LIN {X 0,Y 71.337,Z 768.88,A -85,B 0,C 180,E1 -28289.511,E2 -28289.511} C_VEL
LIN {X 0,Y 69.324,Z 765.278,A -85,B 0,C 180,E1 -28300.962,E2 -28300.962} C_VEL
LIN {X 0,Y 69.422,Z 761.782,A -85,B 0,C 180,E1 -28309.101,E2 -28309.101} C_VEL
LIN {X 0,Y 70.478,Z 757.39,A -85,B 0,C 180,E1 -28317.054,E2 -28317.054} C_VEL
LIN {X 0,Y 72.906,Z 750.784,A -85,B 0,C 180,E1 -28326.145,E2 -28326.145} C_VEL
LIN {X 0,Y 76.398,Z 743.132,A -85,B 0,C 180,E1 -28333.978,E2 -28333.978} C_VEL
LIN {X 0,Y 79.45,Z 736.76,A -85,B 0,C 180,E1 -28338.96,E2 -28338.96} C_VEL
LIN {X 0,Y 80.091,Z 734.246,A -85,B 0,C 180,E1 -28340.836,E2 -28340.836} C_VEL
LIN {X 0,Y 79.689,Z 730.08,A -85,B 0,C 180,E1 -28344.147,E2 -28344.147} C_VEL
LIN {X 0,Y 79.29,Z 724.776,A -85,B 0,C 180,E1 -28348.027,E2 -28348.027} C_VEL
LIN {X 0,Y 79.728,Z 722.85,A -85,B 0,C 180,E1 -28349.133,E2 -28349.133} C_VEL
LIN {X 0,Y 79.98,Z 721.934,A -85,B 0,C 180,E1 -28349.708,E2 -28349.708} C_VEL
LIN {X 0,Y 74.87,Z 732.271,A -85,B 0,C 180,E1 -28355.384,E2 -28355.384} C_VEL
LIN {X 0,Y 69.732,Z 742.158,A -85,B 0,C 180,E1 -28363.104,E2 -28363.104} C_VEL
LIN {X 0,Y 66.404,Z 748.939,A -85,B 0,C 180,E1 -28370.385,E2 -28370.385} C_VEL
LIN {X 0,Y 63.943,Z 754.671,A -85,B 0,C 180,E1 -28378.444,E2 -28378.444} C_VEL
LIN {X 0,Y 62.32,Z 759.792,A -85,B 0,C 180,E1 -28387.868,E2 -28387.868} C_VEL
LIN {X 0,Y 62.114,Z 763.686,A -85,B 0,C 180,E1 -28397.243,E2 -28397.243} C_VEL
LIN {X 0,Y 63.149,Z 766.579,A -85,B 0,C 180,E1 -28406.188,E2 -28406.188} C_VEL
LIN {X 0,Y 65.509,Z 768.703,A -85,B 0,C 180,E1 -28414.587,E2 -28414.587} C_VEL
LIN {X 0,Y 69.052,Z 770.07,A -85,B 0,C 180,E1 -28422.221,E2 -28422.221} C_VEL
LIN {X 0,Y 73.618,Z 770.772,A -85,B 0,C 180,E1 -28428.993,E2 -28428.993} C_VEL
LIN {X 0,Y 79.004,Z 770.85,A -85,B 0,C 180,E1 -28434.896,E2 -28434.896} C_VEL
LIN {X 0,Y 85.242,Z 770.227,A -85,B 0,C 180,E1 -28440,E2 -28440} C_VEL
LIN {X 0,Y 92.081,Z 768.983,A -85,B 0,C 180,E1 -28444.377,E2 -28444.377} C_VEL
LIN {X 0,Y 103.238,Z 765.801,A -85,B 0,C 180,E1 -28449.799,E2 -28449.799} C_VEL
LIN {X 0,Y 115.295,Z 760.919,A -85,B 0,C 180,E1 -28454.112,E2 -28454.112} C_VEL
LIN {X 0,Y 116.057,Z 760.554,A -85,B 0,C 180,E1 -28454.334,E2 -28454.334} C_VEL
LIN {X 0,Y 116.658,Z 760.204,A -85,B 0,C 180,E1 -28455.446,E2 -28455.446} C_VEL
LIN {X 0,Y 117.087,Z 759.92,A -85,B 0,C 180,E1 -28457.465,E2 -28457.465} C_VEL
LIN {X 0,Y 117.189,Z 759.909,A -85,B 0,C 180,E1 -28461.09,E2 -28461.09} C_VEL
LIN {X 0,Y 116.912,Z 760.433,A -85,B 0,C 180,E1 -28465.621,E2 -28465.621} C_VEL
LIN {X 0,Y 115.494,Z 761.467,A -85,B 0,C 180,E1 -28468.077,E2 -28468.077} C_VEL
LIN {X 0,Y 106.748,Z 765.452,A -85,B 0,C 180,E1 -28471.146,E2 -28471.146} C_VEL
LIN {X 0,Y 95.397,Z 769.456,A -85,B 0,C 180,E1 -28475.87,E2 -28475.87} C_VEL
LIN {X 0,Y 85.175,Z 771.953,A -85,B 0,C 180,E1 -28482.049,E2 -28482.049} C_VEL
LIN {X 0,Y 76.217,Z 773.061,A -85,B 0,C 180,E1 -28489.802,E2 -28489.802} C_VEL
LIN {X 0,Y 69.092,Z 772.817,A -85,B 0,C 180,E1 -28499.432,E2 -28499.432} C_VEL
LIN {X 0,Y 64.622,Z 771.167,A -85,B 0,C 180,E1 -28510.96,E2 -28510.96} C_VEL
LIN {X 0,Y 63.47,Z 769.803,A -85,B 0,C 180,E1 -28517.208,E2 -28517.208} C_VEL
LIN {X 0,Y 63.081,Z 766.419,A -85,B 0,C 180,E1 -28529.205,E2 -28529.205} C_VEL
LIN {X 0,Y 62.97,Z 768.91,A -85,B 0,C 180,E1 -28536.411,E2 -28536.411} C_VEL
LIN {X 0,Y 64.724,Z 772.076,A -85,B 0,C 180,E1 -28549.014,E2 -28549.014} C_VEL
LIN {X 0,Y 69.121,Z 773.803,A -85,B 0,C 180,E1 -28560.559,E2 -28560.559} C_VEL
LIN {X 0,Y 76.278,Z 774.156,A -85,B 0,C 180,E1 -28570.165,E2 -28570.165} C_VEL
LIN {X 0,Y 85.222,Z 773.146,A -85,B 0,C 180,E1 -28577.922,E2 -28577.922} C_VEL
LIN {X 0,Y 95.403,Z 770.811,A -85,B 0,C 180,E1 -28584.13,E2 -28584.13} C_VEL
LIN {X 0,Y 106.73,Z 767.014,A -85,B 0,C 180,E1 -28588.876,E2 -28588.876} C_VEL
LIN {X 0,Y 112.602,Z 764.525,A -85,B 0,C 180,E1 -28590.906,E2 -28590.906} C_VEL
LIN {X 0,Y 114.05,Z 763.44,A -85,B 0,C 180,E1 -28594.447,E2 -28594.447} C_VEL
LIN {X 0,Y 114.945,Z 762.708,A -85,B 0,C 180,E1 -28598.478,E2 -28598.478} C_VEL
LIN {X 0,Y 115.002,Z 762.636,A -85,B 0,C 180,E1 -28602.208,E2 -28602.208} C_VEL
LIN {X 0,Y 113.563,Z 763.347,A -85,B 0,C 180,E1 -28605.668,E2 -28605.668} C_VEL
LIN {X 0,Y 105.528,Z 766.471,A -85,B 0,C 180,E1 -28608.475,E2 -28608.475} C_VEL
LIN {X 0,Y 97.929,Z 768.816,A -85,B 0,C 180,E1 -28611.748,E2 -28611.748} C_VEL
LIN {X 0,Y 90.768,Z 770.452,A -85,B 0,C 180,E1 -28615.559,E2 -28615.559} C_VEL
LIN {X 0,Y 84.136,Z 771.476,A -85,B 0,C 180,E1 -28620,E2 -28620} C_VEL
LIN {X 0,Y 77.686,Z 771.834,A -85,B 0,C 180,E1 -28625.639,E2 -28625.639} C_VEL
LIN {X 0,Y 71.968,Z 771.456,A -85,B 0,C 180,E1 -28632.425,E2 -28632.425} C_VEL
LIN {X 0,Y 67.426,Z 770.313,A -85,B 0,C 180,E1 -28640.26,E2 -28640.26} C_VEL
LIN {X 0,Y 64.225,Z 768.384,A -85,B 0,C 180,E1 -28648.901,E2 -28648.901} C_VEL
LIN {X 0,Y 62.494,Z 765.631,A -85,B 0,C 180,E1 -28658.07,E2 -28658.07} C_VEL
LIN {X 0,Y 62.385,Z 760.987,A -85,B 0,C 180,E1 -28669.854,E2 -28669.854} C_VEL
LIN {X 0,Y 63.683,Z 756.191,A -85,B 0,C 180,E1 -28678.955,E2 -28678.955} C_VEL
LIN {X 0,Y 66.102,Z 750.18,A -85,B 0,C 180,E1 -28687.728,E2 -28687.728} C_VEL
LIN {X 0,Y 69.435,Z 743.283,A -85,B 0,C 180,E1 -28695.34,E2 -28695.34} C_VEL
LIN {X 0,Y 73.981,Z 734.44,A -85,B 0,C 180,E1 -28702.492,E2 -28702.492} C_VEL
LIN {X 0,Y 78.93,Z 724.628,A -85,B 0,C 180,E1 -28708.238,E2 -28708.238} C_VEL
LIN {X 0,Y 79.728,Z 722.85,A -85,B 0,C 180,E1 -28709.133,E2 -28709.133} C_VEL
LIN {X 0,Y 79.709,Z 722.855,A -85,B 0,C 180,E1 -28709.872,E2 -28709.872} C_VEL
LIN {X 0,Y 79.088,Z 724.397,A -85,B 0,C 180,E1 -28711,E2 -28711} C_VEL
LIN {X 0,Y 76.998,Z 727.904,A -85,B 0,C 180,E1 -28712.689,E2 -28712.689} C_VEL
LIN {X 0,Y 73.455,Z 731.935,A -85,B 0,C 180,E1 -28714.61,E2 -28714.61} C_VEL
LIN {X 0,Y 65.764,Z 739.297,A -85,B 0,C 180,E1 -28718.654,E2 -28718.654} C_VEL
LIN {X 0,Y 62.667,Z 742.696,A -85,B 0,C 180,E1 -28721.828,E2 -28721.828} C_VEL
LIN {X 0,Y 62.236,Z 743.403,A -85,B 0,C 180,E1 -28722.578,E2 -28722.578} C_VEL
LIN {X 0,Y 58.745,Z 750.185,A -85,B 0,C 180,E1 -28731.03,E2 -28731.03} C_VEL
LIN {X 0,Y 55.942,Z 756.755,A -85,B 0,C 180,E1 -28742.267,E2 -28742.267} C_VEL
LIN {X 0,Y 54.973,Z 762.068,A -85,B 0,C 180,E1 -28754.67,E2 -28754.67} C_VEL
LIN {X 0,Y 55.83,Z 765.581,A -85,B 0,C 180,E1 -28765.499,E2 -28765.499} C_VEL
LIN {X 0,Y 59.978,Z 769.007,A -85,B 0,C 180,E1 -28779.613,E2 -28779.613} C_VEL
LIN {X 0,Y 64.646,Z 770.427,A -85,B 0,C 180,E1 -28788.067,E2 -28788.067} C_VEL
LIN {X 0,Y 70.51,Z 771.064,A -85,B 0,C 180,E1 -28795.341,E2 -28795.341} C_VEL
LIN {X 0,Y 77.327,Z 770.958,A -85,B 0,C 180,E1 -28801.394,E2 -28801.394} C_VEL
LIN {X 0,Y 84.851,Z 770.124,A -85,B 0,C 180,E1 -28806.334,E2 -28806.334} C_VEL
LIN {X 0,Y 92.897,Z 768.516,A -85,B 0,C 180,E1 -28810.435,E2 -28810.435} C_VEL
LIN {X 0,Y 101.332,Z 766.144,A -85,B 0,C 180,E1 -28813.844,E2 -28813.844} C_VEL
LIN {X 0,Y 110.025,Z 762.999,A -85,B 0,C 180,E1 -28816.642,E2 -28816.642} C_VEL
LIN {X 0,Y 110.54,Z 762.772,A -85,B 0,C 180,E1 -28817.514,E2 -28817.514} C_VEL
LIN {X 0,Y 110.567,Z 762.896,A -85,B 0,C 180,E1 -28822.419,E2 -28822.419} C_VEL
LIN {X 0,Y 109.348,Z 763.697,A -85,B 0,C 180,E1 -28825.871,E2 -28825.871} C_VEL
LIN {X 0,Y 100.245,Z 767.168,A -85,B 0,C 180,E1 -28828.799,E2 -28828.799} C_VEL
LIN {X 0,Y 91.428,Z 769.791,A -85,B 0,C 180,E1 -28832.272,E2 -28832.272} C_VEL
LIN {X 0,Y 80.584,Z 772.023,A -85,B 0,C 180,E1 -28838.291,E2 -28838.291} C_VEL
LIN {X 0,Y 70.924,Z 772.909,A -85,B 0,C 180,E1 -28846.084,E2 -28846.084} C_VEL
LIN {X 0,Y 63.07,Z 772.384,A -85,B 0,C 180,E1 -28856.144,E2 -28856.144} C_VEL
LIN {X 0,Y 57.958,Z 770.51,A -85,B 0,C 180,E1 -28868.671,E2 -28868.671} C_VEL
LIN {X 0,Y 56.601,Z 769.057,A -85,B 0,C 180,E1 -28875.624,E2 -28875.624} C_VEL
LIN {X 0,Y 56.083,Z 765.346,A -85,B 0,C 180,E1 -28889.106,E2 -28889.106} C_VEL
LIN {X 0,Y 55.97,Z 768.007,A -85,B 0,C 180,E1 -28897.217,E2 -28897.217} C_VEL
LIN {X 0,Y 56.623,Z 769.911,A -85,B 0,C 180,E1 -28904.376,E2 -28904.376} C_VEL
LIN {X 0,Y 60.188,Z 772.525,A -85,B 0,C 180,E1 -28917.847,E2 -28917.847} C_VEL
LIN {X 0,Y 66.808,Z 773.802,A -85,B 0,C 180,E1 -28929.14,E2 -28929.14} C_VEL
LIN {X 0,Y 75.603,Z 773.75,A -85,B 0,C 180,E1 -28938.048,E2 -28938.048} C_VEL
LIN {X 0,Y 85.892,Z 772.333,A -85,B 0,C 180,E1 -28944.912,E2 -28944.912} C_VEL
LIN {X 0,Y 97.253,Z 769.539,A -85,B 0,C 180,E1 -28950.136,E2 -28950.136} C_VEL
LIN {X 0,Y 106.304,Z 766.519,A -85,B 0,C 180,E1 -28953.193,E2 -28953.193} C_VEL
LIN {X 0,Y 107.731,Z 765.731,A -85,B 0,C 180,E1 -28955.971,E2 -28955.971} C_VEL
LIN {X 0,Y 108.018,Z 765.544,A -85,B 0,C 180,E1 -28957.022,E2 -28957.022} C_VEL
LIN {X 0,Y 108.329,Z 765.267,A -85,B 0,C 180,E1 -28961.072,E2 -28961.072} C_VEL
LIN {X 0,Y 107.845,Z 765.438,A -85,B 0,C 180,E1 -28962.947,E2 -28962.947} C_VEL
LIN {X 0,Y 101.776,Z 767.468,A -85,B 0,C 180,E1 -28965.189,E2 -28965.189} C_VEL
LIN {X 0,Y 93.203,Z 769.734,A -85,B 0,C 180,E1 -28968.607,E2 -28968.607} C_VEL
LIN {X 0,Y 81.279,Z 771.719,A -85,B 0,C 180,E1 -28975.04,E2 -28975.04} C_VEL
LIN {X 0,Y 74.635,Z 772.074,A -85,B 0,C 180,E1 -28980,E2 -28980} C_VEL
LIN {X 0,Y 68.707,Z 771.862,A -85,B 0,C 180,E1 -28985.871,E2 -28985.871} C_VEL
LIN {X 0,Y 63.649,Z 770.982,A -85,B 0,C 180,E1 -28992.758,E2 -28992.758} C_VEL
LIN {X 0,Y 57.995,Z 768.511,A -85,B 0,C 180,E1 -29005.097,E2 -29005.097} C_VEL
LIN {X 0,Y 55.23,Z 764.137,A -85,B 0,C 180,E1 -29020.223,E2 -29020.223} C_VEL
LIN {X 0,Y 55.62,Z 759.061,A -85,B 0,C 180,E1 -29033.115,E2 -29033.115} C_VEL
LIN {X 0,Y 57.844,Z 752.738,A -85,B 0,C 180,E1 -29044.83,E2 -29044.83} C_VEL
LIN {X 0,Y 61.613,Z 745.011,A -85,B 0,C 180,E1 -29055.126,E2 -29055.126} C_VEL
LIN {X 0,Y 66.169,Z 736.739,A -85,B 0,C 180,E1 -29063.005,E2 -29063.005} C_VEL
LIN {X 0,Y 71.341,Z 727.085,A -85,B 0,C 180,E1 -29069.575,E2 -29069.575} C_VEL
LIN {X 0,Y 65.022,Z 738.266,A -85,B 0,C 180,E1 -29077.615,E2 -29077.615} C_VEL
LIN {X 0,Y 62.236,Z 743.403,A -85,B 0,C 180,E1 -29082.578,E2 -29082.578} C_VEL
LIN {X 0,Y 59.725,Z 746.862,A -85,B 0,C 180,E1 -29086.416,E2 -29086.416} C_VEL
LIN {X 0,Y 54.307,Z 751.878,A -85,B 0,C 180,E1 -29093.106,E2 -29093.106} C_VEL
LIN {X 0,Y 49.514,Z 756.287,A -85,B 0,C 180,E1 -29101.51,E2 -29101.51} C_VEL
LIN {X 0,Y 48.175,Z 758.808,A -85,B 0,C 180,E1 -29107.661,E2 -29107.661} C_VEL
LIN {X 0,Y 48.163,Z 763.325,A -85,B 0,C 180,E1 -29120.915,E2 -29120.915} C_VEL
LIN {X 0,Y 50.899,Z 767.174,A -85,B 0,C 180,E1 -29135.529,E2 -29135.529} C_VEL
LIN {X 0,Y 57.195,Z 769.99,A -85,B 0,C 180,E1 -29149.408,E2 -29149.408} C_VEL
LIN {X 0,Y 65.904,Z 771.234,A -85,B 0,C 180,E1 -29160,E2 -29160} C_VEL
LIN {X 0,Y 72.751,Z 771.307,A -85,B 0,C 180,E1 -29165.543,E2 -29165.543} C_VEL
LIN {X 0,Y 80.268,Z 770.682,A -85,B 0,C 180,E1 -29170.085,E2 -29170.085} C_VEL
LIN {X 0,Y 88.229,Z 769.438,A -85,B 0,C 180,E1 -29173.826,E2 -29173.826} C_VEL
LIN {X 0,Y 100.893,Z 766.228,A -85,B 0,C 180,E1 -29178.268,E2 -29178.268} C_VEL
LIN {X 0,Y 103.865,Z 765.283,A -85,B 0,C 180,E1 -29179.775,E2 -29179.775} C_VEL
LIN {X 0,Y 103.031,Z 765.767,A -85,B 0,C 180,E1 -29183.41,E2 -29183.41} C_VEL
LIN {X 0,Y 93.933,Z 768.591,A -85,B 0,C 180,E1 -29186.131,E2 -29186.131} C_VEL
LIN {X 0,Y 81.977,Z 771.274,A -85,B 0,C 180,E1 -29190.989,E2 -29190.989} C_VEL
LIN {X 0,Y 71.017,Z 772.534,A -85,B 0,C 180,E1 -29197.66,E2 -29197.66} C_VEL
LIN {X 0,Y 61.386,Z 772.456,A -85,B 0,C 180,E1 -29206.617,E2 -29206.617} C_VEL
LIN {X 0,Y 53.982,Z 771.053,A -85,B 0,C 180,E1 -29218.62,E2 -29218.62} C_VEL
LIN {X 0,Y 49.792,Z 768.227,A -85,B 0,C 180,E1 -29233.606,E2 -29233.606} C_VEL
LIN {X 0,Y 49.059,Z 764.257,A -85,B 0,C 180,E1 -29248.977,E2 -29248.977} C_VEL
LIN {X 0,Y 49.273,Z 768.08,A -85,B 0,C 180,E1 -29262.358,E2 -29262.358} C_VEL
LIN {X 0,Y 51.547,Z 770.652,A -85,B 0,C 180,E1 -29274.147,E2 -29274.147} C_VEL
LIN {X 0,Y 57.339,Z 772.841,A -85,B 0,C 180,E1 -29287.799,E2 -29287.799} C_VEL
LIN {X 0,Y 66.032,Z 773.671,A -85,B 0,C 180,E1 -29298.166,E2 -29298.166} C_VEL
LIN {X 0,Y 76.424,Z 773.189,A -85,B 0,C 180,E1 -29305.862,E2 -29305.862} C_VEL
LIN {X 0,Y 87.853,Z 771.401,A -85,B 0,C 180,E1 -29311.642,E2 -29311.642} C_VEL
LIN {X 0,Y 100.151,Z 768.209,A -85,B 0,C 180,E1 -29315.823,E2 -29315.823} C_VEL
LIN {X 0,Y 101.424,Z 767.598,A -85,B 0,C 180,E1 -29319.729,E2 -29319.729} C_VEL
LIN {X 0,Y 95.025,Z 769.295,A -85,B 0,C 180,E1 -29322.792,E2 -29322.792} C_VEL
LIN {X 0,Y 86.845,Z 770.938,A -85,B 0,C 180,E1 -29325.95,E2 -29325.95} C_VEL
LIN {X 0,Y 78.482,Z 772.013,A -85,B 0,C 180,E1 -29330.088,E2 -29330.088} C_VEL
LIN {X 0,Y 70.519,Z 772.335,A -85,B 0,C 180,E1 -29335.307,E2 -29335.307} C_VEL
LIN {X 0,Y 63.289,Z 771.897,A -85,B 0,C 180,E1 -29341.876,E2 -29341.876} C_VEL
LIN {X 0,Y 57.103,Z 770.711,A -85,B 0,C 180,E1 -29350.051,E2 -29350.051} C_VEL
LIN {X 0,Y 52.295,Z 768.758,A -85,B 0,C 180,E1 -29359.816,E2 -29359.816} C_VEL
LIN {X 0,Y 48.53,Z 764.728,A -85,B 0,C 180,E1 -29375.4,E2 -29375.4} C_VEL
LIN {X 0,Y 48.312,Z 759.538,A -85,B 0,C 180,E1 -29390.899,E2 -29390.899} C_VEL
LIN {X 0,Y 49.928,Z 754.516,A -85,B 0,C 180,E1 -29402.167,E2 -29402.167} C_VEL
LIN {X 0,Y 52.932,Z 748.24,A -85,B 0,C 180,E1 -29412.732,E2 -29412.732} C_VEL
LIN {X 0,Y 56.893,Z 741.334,A -85,B 0,C 180,E1 -29421.211,E2 -29421.211} C_VEL
LIN {X 0,Y 62.327,Z 732.188,A -85,B 0,C 180,E1 -29429.19,E2 -29429.19} C_VEL
LIN {X 0,Y 62.459,Z 731.607,A -85,B 0,C 180,E1 -29429.695,E2 -29429.695} C_VEL
LIN {X 0,Y 56.769,Z 741.056,A -85,B 0,C 180,E1 -29437.943,E2 -29437.943} C_VEL
LIN {X 0,Y 52.618,Z 748.32,A -85,B 0,C 180,E1 -29447.078,E2 -29447.078} C_VEL
LIN {X 0,Y 49.654,Z 754.427,A -85,B 0,C 180,E1 -29457.657,E2 -29457.657} C_VEL
LIN {X 0,Y 48.175,Z 758.808,A -85,B 0,C 180,E1 -29467.661,E2 -29467.661} C_VEL
LIN {X 0,Y 47.291,Z 761.108,A -85,B 0,C 180,E1 -29474.095,E2 -29474.095} C_VEL
LIN {X 0,Y 45.168,Z 764.209,A -85,B 0,C 180,E1 -29485.486,E2 -29485.486} C_VEL
LIN {X 0,Y 44.6,Z 766.216,A -85,B 0,C 180,E1 -29495.372,E2 -29495.372} C_VEL
LIN {X 0,Y 45.791,Z 767.582,A -85,B 0,C 180,E1 -29502.587,E2 -29502.587} C_VEL
LIN {X 0,Y 46.589,Z 767.975,A -85,B 0,C 180,E1 -29504.783,E2 -29504.783} C_VEL
LIN {X 0,Y 50.283,Z 769.453,A -85,B 0,C 180,E1 -29511.965,E2 -29511.965} C_VEL
LIN {X 0,Y 56.309,Z 770.785,A -85,B 0,C 180,E1 -29520,E2 -29520} C_VEL
LIN {X 0,Y 63.702,Z 771.488,A -85,B 0,C 180,E1 -29526.839,E2 -29526.839} C_VEL
LIN {X 0,Y 71.882,Z 771.482,A -85,B 0,C 180,E1 -29532.132,E2 -29532.132} C_VEL
LIN {X 0,Y 80.513,Z 770.74,A -85,B 0,C 180,E1 -29536.23,E2 -29536.23} C_VEL
LIN {X 0,Y 93.557,Z 768.356,A -85,B 0,C 180,E1 -29540.773,E2 -29540.773} C_VEL
LIN {X 0,Y 91.035,Z 769.034,A -85,B 0,C 180,E1 -29542.123,E2 -29542.123} C_VEL
LIN {X 0,Y 78.205,Z 771.424,A -85,B 0,C 180,E1 -29546.701,E2 -29546.701} C_VEL
LIN {X 0,Y 66.915,Z 772.393,A -85,B 0,C 180,E1 -29552.841,E2 -29552.841} C_VEL
LIN {X 0,Y 56.43,Z 772.081,A -85,B 0,C 180,E1 -29561.651,E2 -29561.651} C_VEL
LIN {X 0,Y 48.067,Z 770.39,A -85,B 0,C 180,E1 -29574.213,E2 -29574.213} C_VEL
LIN {X 0,Y 43.066,Z 767.342,A -85,B 0,C 180,E1 -29590.955,E2 -29590.955} C_VEL
LIN {X 0,Y 42.062,Z 763.107,A -85,B 0,C 180,E1 -29609.107,E2 -29609.107} C_VEL
LIN {X 0,Y 42.451,Z 767.071,A -85,B 0,C 180,E1 -29624.383,E2 -29624.383} C_VEL
LIN {X 0,Y 45.185,Z 769.845,A -85,B 0,C 180,E1 -29637.819,E2 -29637.819} C_VEL
LIN {X 0,Y 51.915,Z 772.252,A -85,B 0,C 180,E1 -29652.604,E2 -29652.604} C_VEL
LIN {X 0,Y 61.512,Z 773.376,A -85,B 0,C 180,E1 -29663.113,E2 -29663.113} C_VEL
LIN {X 0,Y 72.664,Z 773.155,A -85,B 0,C 180,E1 -29670.518,E2 -29670.518} C_VEL
LIN {X 0,Y 84.71,Z 771.614,A -85,B 0,C 180,E1 -29675.874,E2 -29675.874} C_VEL
LIN {X 0,Y 91.037,Z 770.341,A -85,B 0,C 180,E1 -29677.884,E2 -29677.884} C_VEL
LIN {X 0,Y 91.711,Z 770.148,A -85,B 0,C 180,E1 -29678.976,E2 -29678.976} C_VEL
LIN {X 0,Y 80.944,Z 771.87,A -85,B 0,C 180,E1 -29682.767,E2 -29682.767} C_VEL
LIN {X 0,Y 69.678,Z 772.571,A -85,B 0,C 180,E1 -29688.362,E2 -29688.362} C_VEL
LIN {X 0,Y 62.293,Z 772.356,A -85,B 0,C 180,E1 -29693.522,E2 -29693.522} C_VEL
LIN {X 0,Y 55.626,Z 771.484,A -85,B 0,C 180,E1 -29700,E2 -29700} C_VEL
LIN {X 0,Y 47.331,Z 769.062,A -85,B 0,C 180,E1 -29712.865,E2 -29712.865} C_VEL
LIN {X 0,Y 42.117,Z 765.069,A -85,B 0,C 180,E1 -29730.04,E2 -29730.04} C_VEL
LIN {X 0,Y 41.042,Z 760.339,A -85,B 0,C 180,E1 -29746.762,E2 -29746.762} C_VEL
LIN {X 0,Y 42.86,Z 754.21,A -85,B 0,C 180,E1 -29763.085,E2 -29763.085} C_VEL
LIN {X 0,Y 46.853,Z 746.667,A -85,B 0,C 180,E1 -29776.993,E2 -29776.993} C_VEL
LIN {X 0,Y 52.098,Z 738.445,A -85,B 0,C 180,E1 -29787.097,E2 -29787.097} C_VEL
LIN {X 0,Y 53.573,Z 735.891,A -85,B 0,C 180,E1 -29789.644,E2 -29789.644} C_VEL
LIN {X 0,Y 47.44,Z 745.332,A -85,B 0,C 180,E1 -29800.668,E2 -29800.668} C_VEL
LIN {X 0,Y 43.137,Z 752.896,A -85,B 0,C 180,E1 -29814.026,E2 -29814.026} C_VEL
LIN {X 0,Y 41.104,Z 758.218,A -85,B 0,C 180,E1 -29827.429,E2 -29827.429} C_VEL
LIN {X 0,Y 41.207,Z 762.766,A -85,B 0,C 180,E1 -29842.434,E2 -29842.434} C_VEL
LIN {X 0,Y 44.814,Z 767.053,A -85,B 0,C 180,E1 -29860.201,E2 -29860.201} C_VEL
LIN {X 0,Y 46.589,Z 767.975,A -85,B 0,C 180,E1 -29864.783,E2 -29864.783} C_VEL
LIN {X 0,Y 48.975,Z 769.19,A -85,B 0,C 180,E1 -29871.131,E2 -29871.131} C_VEL
LIN {X 0,Y 52.656,Z 770.583,A -85,B 0,C 180,E1 -29881.425,E2 -29881.425} C_VEL
LIN {X 0,Y 57.846,Z 771.468,A -85,B 0,C 180,E1 -29890.173,E2 -29890.173} C_VEL
LIN {X 0,Y 62.271,Z 771.718,A -85,B 0,C 180,E1 -29893.91,E2 -29893.91} C_VEL
LIN {X 0,Y 74.711,Z 771.494,A -85,B 0,C 180,E1 -29899.839,E2 -29899.839} C_VEL
LIN {X 0,Y 76.324,Z 771.354,A -85,B 0,C 180,E1 -29900.459,E2 -29900.459} C_VEL
LIN {X 0,Y 75.649,Z 771.48,A -85,B 0,C 180,E1 -29901.724,E2 -29901.724} C_VEL
LIN {X 0,Y 63.346,Z 772.205,A -85,B 0,C 180,E1 -29907.438,E2 -29907.438} C_VEL
LIN {X 0,Y 51.978,Z 771.6,A -85,B 0,C 180,E1 -29915.786,E2 -29915.786} C_VEL
LIN {X 0,Y 42.518,Z 769.694,A -85,B 0,C 180,E1 -29928.616,E2 -29928.616} C_VEL
LIN {X 0,Y 36.469,Z 766.397,A -85,B 0,C 180,E1 -29947.335,E2 -29947.335} C_VEL
LIN {X 0,Y 35.095,Z 761.855,A -85,B 0,C 180,E1 -29968.929,E2 -29968.929} C_VEL
LIN {X 0,Y 35.692,Z 766.026,A -85,B 0,C 180,E1 -29987.184,E2 -29987.184} C_VEL
LIN {X 0,Y 39.071,Z 768.979,A -85,B 0,C 180,E1 -30002.664,E2 -30002.664} C_VEL
LIN {X 0,Y 46.942,Z 771.641,A -85,B 0,C 180,E1 -30018.473,E2 -30018.473} C_VEL
LIN {X 0,Y 57.525,Z 772.985,A -85,B 0,C 180,E1 -30028.788,E2 -30028.788} C_VEL
LIN {X 0,Y 69.436,Z 773.042,A -85,B 0,C 180,E1 -30035.641,E2 -30035.641} C_VEL
LIN {X 0,Y 75.667,Z 772.586,A -85,B 0,C 180,E1 -30038.255,E2 -30038.255} C_VEL
LIN {X 0,Y 75.211,Z 772.581,A -85,B 0,C 180,E1 -30039.143,E2 -30039.143} C_VEL
LIN {X 0,Y 66.079,Z 772.839,A -85,B 0,C 180,E1 -30043.187,E2 -30043.187} C_VEL
LIN {X 0,Y 57.351,Z 772.312,A -85,B 0,C 180,E1 -30048.636,E2 -30048.636} C_VEL
LIN {X 0,Y 46.119,Z 770.28,A -85,B 0,C 180,E1 -30060,E2 -30060} C_VEL
LIN {X 0,Y 40.383,Z 768.155,A -85,B 0,C 180,E1 -30070.023,E2 -30070.023} C_VEL
LIN {X 0,Y 35.054,Z 764.021,A -85,B 0,C 180,E1 -30088.805,E2 -30088.805} C_VEL
LIN {X 0,Y 33.957,Z 760.018,A -85,B 0,C 180,E1 -30105,E2 -30105} C_VEL
LIN {X 0,Y 35.772,Z 753.922,A -85,B 0,C 180,E1 -30124.298,E2 -30124.298} C_VEL
LIN {X 0,Y 40.043,Z 746.558,A -85,B 0,C 180,E1 -30139.887,E2 -30139.887} C_VEL
LIN {X 0,Y 44.771,Z 739.789,A -85,B 0,C 180,E1 -30149.408,E2 -30149.408} C_VEL
LIN {X 0,Y 44.462,Z 739.806,A -85,B 0,C 180,E1 -30149.996,E2 -30149.996} C_VEL
LIN {X 0,Y 39.635,Z 746.804,A -85,B 0,C 180,E1 -30160.209,E2 -30160.209} C_VEL
LIN {X 0,Y 35.414,Z 753.873,A -85,B 0,C 180,E1 -30175.812,E2 -30175.812} C_VEL
LIN {X 0,Y 33.8,Z 759.737,A -85,B 0,C 180,E1 -30194.998,E2 -30194.998} C_VEL
LIN {X 0,Y 36.313,Z 764.964,A -85,B 0,C 180,E1 -30217.227,E2 -30217.227} C_VEL
LIN {X 0,Y 42.44,Z 768.392,A -85,B 0,C 180,E1 -30233.474,E2 -30233.474} C_VEL
LIN {X 0,Y 49.27,Z 770.27,A -85,B 0,C 180,E1 -30243.206,E2 -30243.206} C_VEL
LIN {X 0,Y 61.226,Z 771.689,A -85,B 0,C 180,E1 -30253.272,E2 -30253.272} C_VEL
LIN {X 0,Y 62.271,Z 771.718,A -85,B 0,C 180,E1 -30253.91,E2 -30253.91} C_VEL
LIN {X 0,Y 62.87,Z 771.786,A -85,B 0,C 180,E1 -30255.096,E2 -30255.096} C_VEL
LIN {X 0,Y 62.2,Z 771.855,A -85,B 0,C 180,E1 -30257.454,E2 -30257.454} C_VEL
LIN {X 0,Y 59.293,Z 771.905,A -85,B 0,C 180,E1 -30260.851,E2 -30260.851} C_VEL
LIN {X 0,Y 56.525,Z 771.812,A -85,B 0,C 180,E1 -30263.087,E2 -30263.087} C_VEL
LIN {X 0,Y 47.442,Z 771.011,A -85,B 0,C 180,E1 -30269.698,E2 -30269.698} C_VEL
LIN {X 0,Y 39.105,Z 769.339,A -85,B 0,C 180,E1 -30278.85,E2 -30278.85} C_VEL
LIN {X 0,Y 33.226,Z 767.309,A -85,B 0,C 180,E1 -30290.62,E2 -30290.62} C_VEL
LIN {X 0,Y 28.315,Z 763.018,A -85,B 0,C 180,E1 -30315.635,E2 -30315.635} C_VEL
LIN {X 0,Y 28.117,Z 760.526,A -85,B 0,C 180,E1 -30328.887,E2 -30328.887} C_VEL
LIN {X 0,Y 29.072,Z 764.865,A -85,B 0,C 180,E1 -30351.267,E2 -30351.267} C_VEL
LIN {X 0,Y 33.34,Z 768.019,A -85,B 0,C 180,E1 -30369.233,E2 -30369.233} C_VEL
LIN {X 0,Y 42.578,Z 770.94,A -85,B 0,C 180,E1 -30385.626,E2 -30385.626} C_VEL
LIN {X 0,Y 54.183,Z 772.579,A -85,B 0,C 180,E1 -30395.232,E2 -30395.232} C_VEL
LIN {X 0,Y 60.429,Z 772.903,A -85,B 0,C 180,E1 -30398.505,E2 -30398.505} C_VEL
LIN {X 0,Y 51.167,Z 771.946,A -85,B 0,C 180,E1 -30404.056,E2 -30404.056} C_VEL
LIN {X 0,Y 42.623,Z 770.264,A -85,B 0,C 180,E1 -30411.642,E2 -30411.642} C_VEL
LIN {X 0,Y 33.136,Z 766.851,A -85,B 0,C 180,E1 -30427.143,E2 -30427.143} C_VEL
LIN {X 0,Y 27.605,Z 762.098,A -85,B 0,C 180,E1 -30450.61,E2 -30450.61} C_VEL
LIN {X 0,Y 27.367,Z 756.542,A -85,B 0,C 180,E1 -30475.408,E2 -30475.408} C_VEL
LIN {X 0,Y 30.372,Z 750.746,A -85,B 0,C 180,E1 -30494.136,E2 -30494.136} C_VEL
LIN {X 0,Y 35.803,Z 743.263,A -85,B 0,C 180,E1 -30509.417,E2 -30509.417} C_VEL
LIN {X 0,Y 35.595,Z 743.185,A -85,B 0,C 180,E1 -30509.995,E2 -30509.995} C_VEL
LIN {X 0,Y 30.674,Z 749.725,A -85,B 0,C 180,E1 -30523.239,E2 -30523.239} C_VEL
LIN {X 0,Y 27.452,Z 755.341,A -85,B 0,C 180,E1 -30540.791,E2 -30540.791} C_VEL
LIN {X 0,Y 26.927,Z 760.119,A -85,B 0,C 180,E1 -30561.525,E2 -30561.525} C_VEL
LIN {X 0,Y 31.249,Z 765.217,A -85,B 0,C 180,E1 -30587.002,E2 -30587.002} C_VEL
LIN {X 0,Y 36.98,Z 767.871,A -85,B 0,C 180,E1 -30600,E2 -30600} C_VEL
LIN {X 0,Y 44.067,Z 769.879,A -85,B 0,C 180,E1 -30609.177,E2 -30609.177} C_VEL
LIN {X 0,Y 51.911,Z 771.208,A -85,B 0,C 180,E1 -30615.71,E2 -30615.71} C_VEL
LIN {X 0,Y 60.284,Z 771.914,A -85,B 0,C 180,E1 -30620.471,E2 -30620.471} C_VEL
LIN {X 0,Y 60.405,Z 771.948,A -85,B 0,C 180,E1 -30621.451,E2 -30621.451} C_VEL
LIN {X 0,Y 48.169,Z 771.111,A -85,B 0,C 180,E1 -30628.914,E2 -30628.914} C_VEL
LIN {X 0,Y 39.105,Z 769.339,A -85,B 0,C 180,E1 -30638.85,E2 -30638.85} C_VEL
LIN {X 0,Y 34.883,Z 768.12,A -85,B 0,C 180,E1 -30644.943,E2 -30644.943} C_VEL
LIN {X 0,Y 27.785,Z 765.247,A -85,B 0,C 180,E1 -30656.491,E2 -30656.491} C_VEL
LIN {X 0,Y 23.137,Z 762.402,A -85,B 0,C 180,E1 -30669.71,E2 -30669.71} C_VEL
LIN {X 0,Y 21.175,Z 759.166,A -85,B 0,C 180,E1 -30687.923,E2 -30687.923} C_VEL
LIN {X 0,Y 22.692,Z 763.667,A -85,B 0,C 180,E1 -30717.69,E2 -30717.69} C_VEL
LIN {X 0,Y 28.224,Z 767.012,A -85,B 0,C 180,E1 -30738.341,E2 -30738.341} C_VEL
LIN {X 0,Y 39.023,Z 770.183,A -85,B 0,C 180,E1 -30754.231,E2 -30754.231} C_VEL
LIN {X 0,Y 41.007,Z 770.576,A -85,B 0,C 180,E1 -30755.835,E2 -30755.835} C_VEL
LIN {X 0,Y 43.742,Z 771.041,A -85,B 0,C 180,E1 -30759.357,E2 -30759.357} C_VEL
LIN {X 0,Y 31.015,Z 767.502,A -85,B 0,C 180,E1 -30772.454,E2 -30772.454} C_VEL
LIN {X 0,Y 22.09,Z 762.593,A -85,B 0,C 180,E1 -30797.331,E2 -30797.331} C_VEL
LIN {X 0,Y 20.074,Z 756.678,A -85,B 0,C 180,E1 -30832.206,E2 -30832.206} C_VEL
LIN {X 0,Y 23.194,Z 750.926,A -85,B 0,C 180,E1 -30857.041,E2 -30857.041} C_VEL
LIN {X 0,Y 25.583,Z 747.851,A -85,B 0,C 180,E1 -30866.055,E2 -30866.055} C_VEL
LIN {X 0,Y 26.508,Z 746.375,A -85,B 0,C 180,E1 -30870.231,E2 -30870.231} C_VEL
LIN {X 0,Y 21.702,Z 752.44,A -85,B 0,C 180,E1 -30888.887,E2 -30888.887} C_VEL
LIN {X 0,Y 19.74,Z 757.721,A -85,B 0,C 180,E1 -30915.388,E2 -30915.388} C_VEL
LIN {X 0,Y 22.092,Z 762.162,A -85,B 0,C 180,E1 -30942.6,E2 -30942.6} C_VEL
LIN {X 0,Y 28.121,Z 765.757,A -85,B 0,C 180,E1 -30961.655,E2 -30961.655} C_VEL
LIN {X 0,Y 36.129,Z 768.522,A -85,B 0,C 180,E1 -30973.458,E2 -30973.458} C_VEL
LIN {X 0,Y 45.169,Z 770.506,A -85,B 0,C 180,E1 -30981.015,E2 -30981.015} C_VEL
LIN {X 0,Y 33.235,Z 768.076,A -85,B 0,C 180,E1 -30992.245,E2 -30992.245} C_VEL
LIN {X 0,Y 24.087,Z 764.267,A -85,B 0,C 180,E1 -31014.308,E2 -31014.308} C_VEL
LIN {X 0,Y 21.175,Z 759.166,A -85,B 0,C 180,E1 -31047.923,E2 -31047.923} C_VEL
LIN {X 0,Y 20.617,Z 760.519,A -85,B 0,C 180,E1 -31057.961,E2 -31057.961} C_VEL
LIN {X 0,Y 19.616,Z 761.634,A -85,B 0,C 180,E1 -31068.513,E2 -31068.513} C_VEL
LIN {X 0,Y 19.371,Z 763.932,A -85,B 0,C 180,E1 -31095.993,E2 -31095.993} C_VEL
LIN {X 0,Y 21.497,Z 764.856,A -85,B 0,C 180,E1 -31105.418,E2 -31105.418} C_VEL
LIN {X 0,Y 24.132,Z 765.884,A -85,B 0,C 180,E1 -31110.906,E2 -31110.906} C_VEL
LIN {X 0,Y 27.679,Z 767.03,A -85,B 0,C 180,E1 -31120.189,E2 -31120.189} C_VEL
LIN {X 0,Y 17.591,Z 762.568,A -85,B 0,C 180,E1 -31140.001,E2 -31140.001} C_VEL
LIN {X 0,Y 12.899,Z 756.773,A -85,B 0,C 180,E1 -31185.033,E2 -31185.033} C_VEL
LIN {X 0,Y 16.122,Z 751.043,A -85,B 0,C 180,E1 -31222.633,E2 -31222.633} C_VEL
LIN {X 0,Y 17.391,Z 749.327,A -85,B 0,C 180,E1 -31229.99,E2 -31229.99} C_VEL
LIN {X 0,Y 12.736,Z 756.455,A -85,B 0,C 180,E1 -31274.94,E2 -31274.94} C_VEL
LIN {X 0,Y 17.688,Z 762.157,A -85,B 0,C 180,E1 -31319.999,E2 -31319.999} C_VEL
LIN {X 0,Y 27.945,Z 766.495,A -85,B 0,C 180,E1 -31339.465,E2 -31339.465} C_VEL
LIN {X 0,Y 24.06,Z 765.288,A -85,B 0,C 180,E1 -31348.815,E2 -31348.815} C_VEL
LIN {X 0,Y 15.188,Z 760.445,A -85,B 0,C 180,E1 -31382.448,E2 -31382.448} C_VEL
LIN {X 0,Y 14.216,Z 757.699,A -85,B 0,C 180,E1 -31409.039,E2 -31409.039} C_VEL
LIN {X 0,Y 16.842,Z 762.335,A -85,B 0,C 180,E1 -31448.764,E2 -31448.764} C_VEL
LIN {X 0,Y 21.497,Z 764.856,A -85,B 0,C 180,E1 -31465.418,E2 -31465.418} C_VEL
LIN {X 0,Y 20.09,Z 764.517,A -85,B 0,C 180,E1 -31465.898,E2 -31465.898} C_VEL
LIN {X 0,Y 14.129,Z 762.649,A -85,B 0,C 180,E1 -31456.29,E2 -31456.29} C_VEL
LIN {X 0,Y 8.246,Z 759.927,A -85,B 0,C 180,E1 -31397.154,E2 -31397.154} C_VEL
LIN {X 0,Y 9.825,Z 759.744,A -85,B 0,C 180,E1 -31363.901,E2 -31363.901} C_VEL
LIN {X 0,Y 12.121,Z 760.45,A -85,B 0,C 180,E1 -31346.941,E2 -31346.941} C_VEL
LIN {X 0,Y 13.392,Z 761.013,A -85,B 0,C 180,E1 -31340.789,E2 -31340.789} C_VEL
LIN {X 0,Y 5.765,Z 754.924,A -85,B 0,C 180,E1 -31270.562,E2 -31270.562} C_VEL
LIN {X 0,Y 7.869,Z 752.167,A -85,B 0,C 180,E1 -31229.978,E2 -31229.978} C_VEL
LIN {X 0,Y 7.158,Z 753.17,A -85,B 0,C 180,E1 -31219.074,E2 -31219.074} C_VEL
LIN {X 0,Y 9.757,Z 759.568,A -85,B 0,C 180,E1 -31130.276,E2 -31130.276} C_VEL
LIN {X 0,Y 13.396,Z 761.483,A -85,B 0,C 180,E1 -31118.921,E2 -31118.921} C_VEL
LIN {X 0,Y 11.068,Z 760.351,A -85,B 0,C 180,E1 -31105.056,E2 -31105.056} C_VEL
LIN {X 0,Y 7.338,Z 756.014,A -85,B 0,C 180,E1 -31046.252,E2 -31046.252} C_VEL
LIN {X 0,Y 11.005,Z 759.878,A -85,B 0,C 180,E1 -30994.556,E2 -30994.556} C_VEL
LIN {X 0,Y 12.121,Z 760.45,A -85,B 0,C 180,E1 -30986.941,E2 -30986.941} C_VEL
LIN {X 0,Y 12.121,Z 760.45,A -85,B 0,C 180,E1 -30986.941,E2 -30986.941}

QRS_NEXT_CUT()

QRS_NEXT()
QRS_HOME()

END
